KUKA KRL program: rechazoemsinf.src, rechazoemsinf.dat

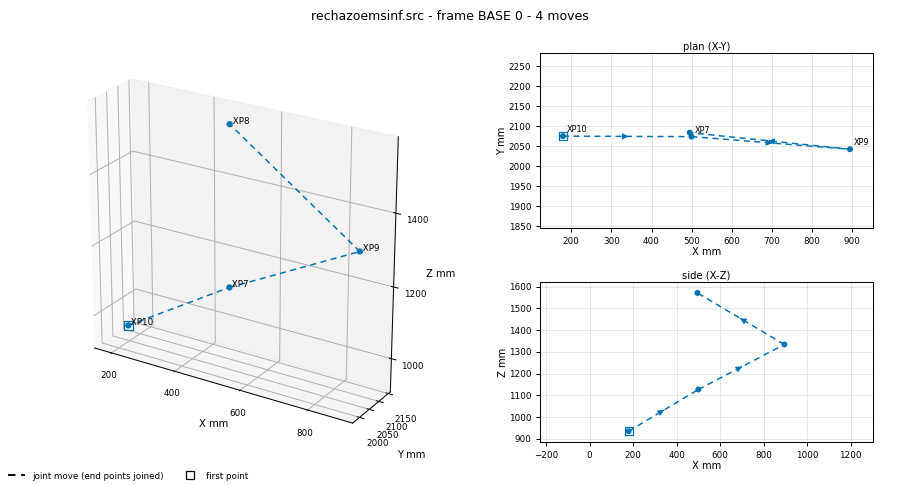
[picture p0: tool path of rechazoemsinf.src in frame BASE 0, 4 of 4 moves have a stored position in this frame; points joined in program order, loops and branches not executed]
--- rechazoemsinf.src ---
&ACCESS RVO1
&REL 33
&COMMENT rechazo ems inferior
&PARAM TEMPLATE = C:\KRC\Roboter\Template\vorgabe
&PARAM EDITMASK = *
DEF RECHAZOEMSINF( )

;================================================
; MODELO   : C-520
; IE GRUPO : 5J
; ESTACION : 85
; ROBOT    : 85r01
; FUNCION  : xxxxxxx
;================================================

;FOLD INI
  ;FOLD BASISTECH INI
    GLOBAL INTERRUPT DECL 3 WHEN $STOPMESS==TRUE DO IR_STOPM ( )
    INTERRUPT ON 3
    BAS (#INITMOV,0 )
  ;ENDFOLD (BASISTECH INI)
;FOLD SPOTTECH INI
;USERSPOT(#INIT)
;ENDFOLD (SPOTTECH INI)
;FOLD GRIPPERTECH INI
USER_GRP(0,DUMMY,DUMMY,GDEFAULT)
INTERRUPT DECL 20 WHEN $FLAG[20]==FALSE DO GRPS(#MON_ERR,20)
;ENDFOLD (GRIPPERTECH INI)
  ;FOLD USER INI
    ;Make your modifications here

  ;ENDFOLD (USER INI)
;ENDFOLD (INI)

I_DATOS_NOK=TRUE

;FOLD PTP P10 CONT Vel=100 % PDAT10 Tool[0] Base[0];%{PE}%R 5.6.13,%MKUKATPBASIS,%CMOVE,%VPTP,%P 1:PTP, 2:P10, 3:C_PTP, 5:100, 7:PDAT10
$BWDSTART=FALSE
PDAT_ACT=PPDAT10
FDAT_ACT=FP10
BAS(#PTP_PARAMS,100)
PTP XP10 C_PTP
;ENDFOLD
;FOLD OUT 18 'LIBERACION AREA 2 ems sup' State=FALSE ;%{PE}%R 5.6.13,%MKUKATPBASIS,%COUT,%VOUTX,%P 2:18, 3:LIBERACION AREA 2 ems sup, 5:FALSE, 6:
$OUT[18]=FALSE
;ENDFOLD
;RECHAZOPOS
;FOLD FORDTECH.Area_Req 4 Safety Position, 0 Return To Home, 0 ;%{PE}%MKUKATPUSER
;Area_Req (4,0,0)

WAIT FOR  ( $IN[20] )
$OUT[20]=FALSE

;ENDFOLD
WAIT SEC 4
;FOLD PTP P7 CONT Vel=30 % PDAT7 Tool[0] Base[0];%{PE}%R 5.6.13,%MKUKATPBASIS,%CMOVE,%VPTP,%P 1:PTP, 2:P7, 3:C_PTP, 5:30, 7:PDAT7
$BWDSTART=FALSE
PDAT_ACT=PPDAT7
FDAT_ACT=FP7
BAS(#PTP_PARAMS,30)
PTP XP7 C_PTP
;ENDFOLD

;FOLD PTP P9 Vel=30 % PDAT9 Tool[0] Base[0];%{PE}%R 5.6.13,%MKUKATPBASIS,%CMOVE,%VPTP,%P 1:PTP, 2:P9, 3:, 5:30, 7:PDAT9
$BWDSTART=FALSE
PDAT_ACT=PPDAT9
FDAT_ACT=FP9
BAS(#PTP_PARAMS,30)
PTP XP9
;ENDFOLD

;FOLD OUT 97 'dedos fuera' State=FALSE ;%{PE}%R 5.6.13,%MKUKATPBASIS,%COUT,%VOUTX,%P 2:97, 3:dedos fuera, 5:FALSE, 6:
$OUT[97]=FALSE
;ENDFOLD
;FOLD OUT 98 'dedos dentro' State=TRUE ;%{PE}%R 5.6.13,%MKUKATPBASIS,%COUT,%VOUTX,%P 2:98, 3:dedos dentro, 5:TRUE, 6:
$OUT[98]=TRUE
;ENDFOLD

;FOLD OUT 89 'pos abrir ip manual' State=TRUE ;%{PE}%R 5.6.13,%MKUKATPBASIS,%COUT,%VOUTX,%P 2:89, 3:pos abrir ip manual, 5:TRUE, 6:
$OUT[89]=TRUE
;ENDFOLD
;FOLD FORDTECH.Tool_Rel 5 ;%{PE}%MKUKATPUSER
TOOL_REL (5)
;ENDFOLD
;FOLD FORDTECH.Tool_Req 5 ;%{PE}%MKUKATPUSER
TOOL_REQ (5)
;ENDFOLD

;FOLD OUT 89 'pos abrir ip manual' State=FALSE ;%{PE}%R 5.6.13,%MKUKATPBASIS,%COUT,%VOUTX,%P 2:89, 3:pos abrir ip manual, 5:FALSE, 6:
$OUT[89]=FALSE
;ENDFOLD
;FOLD OUT 97 'dedos fuera' State=TRUE ;%{PE}%R 5.6.13,%MKUKATPBASIS,%COUT,%VOUTX,%P 2:97, 3:dedos fuera, 5:TRUE, 6:
$OUT[97]=TRUE
;ENDFOLD
;FOLD OUT 98 'dedos dentro' State=FALSE ;%{PE}%R 5.6.13,%MKUKATPBASIS,%COUT,%VOUTX,%P 2:98, 3:dedos dentro, 5:FALSE, 6:
$OUT[98]=FALSE
;ENDFOLD

;FOLD PTP P8 CONT Vel=100 % PDAT8 Tool[0] Base[0];%{PE}%R 5.6.13,%MKUKATPBASIS,%CMOVE,%VPTP,%P 1:PTP, 2:P8, 3:C_PTP, 5:100, 7:PDAT8
$BWDSTART=FALSE
PDAT_ACT=PPDAT8
FDAT_ACT=FP8
BAS(#PTP_PARAMS,100)
PTP XP8 C_PTP
;ENDFOLD
;FOLD FORDTECH.Area_Rel 2 ;%{PE}%MKUKATPUSER
AREA_REL (2)
;ENDFOLD
;FOLD FORDTECH.Area_Rel 3 ;%{PE}%MKUKATPUSER
AREA_REL (3)
;ENDFOLD
;FOLD FORDTECH.Area_Rel 4 ;%{PE}%MKUKATPUSER
AREA_REL (4)
;ENDFOLD
;FOLD FORDTECH.Job_Rdy 4 , 1 ;%{PE}%MKUKATPUSER
JOB_READY (4,1)
;ENDFOLD




END

--- rechazoemsinf.dat ---
&ACCESS RVO1
&REL 33
&COMMENT rechazo ems inferior
&PARAM TEMPLATE = C:\KRC\Roboter\Template\vorgabe
&PARAM EDITMASK = *
DEFDAT  RECHAZOEMSINF
;FOLD EXTERNAL DECLARATIONS;%{PE}%MKUKATPBASIS,%CEXT,%VCOMMON,%P
;FOLD GRIPPERTECH EXT
EXT  H50 (INT  :IN,INT  :IN,INT  :IN,GRP_TYP  :IN )
;ENDFOLD (GRIPPERTECH EXT)
;FOLD SPOTTECH EXT
EXT  USERSPOT (S_COMMAND  :IN,SPOT_TYPE  :IN )
;ENDFOLD (SPOTTECH EXT)
;FOLD BASISTECH EXT;%{PE}%MKUKATPBASIS,%CEXT,%VEXT,%P
EXT  BAS (BAS_COMMAND  :IN,REAL  :IN )
DECL INT SUCCESS
;ENDFOLD (BASISTECH EXT)
;FOLD USER EXT;%{E}%MKUKATPUSER,%CEXT,%VEXT,%P
;Make here your modifications

;ENDFOLD (USER EXT)
;ENDFOLD (EXTERNAL DECLARATIONS)
DECL BASIS_SUGG_T LAST_BASIS={POINT1[] "P10                     ",POINT2[] "P10                     ",CP_PARAMS[] "CPDAT0                  ",PTP_PARAMS[] "PDAT10                  ",CONT[] "C_PTP                   ",CP_VEL[] "2.0                     ",PTP_VEL[] "100                     ",SYNC_PARAMS[] "SYNCDAT                 ",SPL_NAME[] "S0                      "}
DECL PDAT PPDAT0={VEL 100.0,ACC 100.0,APO_DIST 100.0}
DECL E6POS XP0={X 1811.52502,Y -400.592712,Z 796.957886,A -63.3204193,B 28.7300301,C -159.576996,S 2,T 10,E1 0.0,E2 0.0,E3 0.0,E4 0.0,E5 0.0,E6 0.0}
DECL FDAT FP0={TOOL_NO 1,BASE_NO 0,IPO_FRAME #BASE,POINT2[] " ",TQ_STATE FALSE}
DECL PDAT PPDAT1={VEL 100.0,ACC 100.0,APO_DIST 100.0,APO_MODE #CPTP}
DECL E6POS XP1={X 141.040298,Y -131.536896,Z -626.476685,A -0.01522478,B 7.10692596,C 0.110732399,S 2,T 3,E1 0.0,E2 0.0,E3 0.0,E4 0.0,E5 0.0,E6 0.0}
DECL FDAT FP1={TOOL_NO 3,BASE_NO 8,IPO_FRAME #BASE,POINT2[] " ",TQ_STATE FALSE}
DECL PDAT PPDAT2={VEL 100.0,ACC 100.0,APO_DIST 100.0,APO_MODE #CPTP}
DECL E6POS XP2={X 1145.12195,Y 865.575378,Z 1562.22705,A -24.1379299,B -0.725280404,C -90.2146072,S 2,T 2,E1 0.0,E2 0.0,E3 0.0,E4 0.0,E5 0.0,E6 0.0}
DECL FDAT FP2={TOOL_NO 3,BASE_NO 0,IPO_FRAME #BASE,POINT2[] " ",TQ_STATE FALSE}
DECL PDAT PPDAT3={VEL 100.0,ACC 100.0,APO_DIST 100.0,APO_MODE #CPTP}
DECL E6POS XP3={X 1888.578,Y 938.442871,Z 1603.72998,A -59.9518318,B -1.77833796,C -87.043541,S 2,T 2,E1 0.0,E2 0.0,E3 0.0,E4 0.0,E5 0.0,E6 0.0}
DECL FDAT FP3={TOOL_NO 3,BASE_NO 0,IPO_FRAME #BASE,POINT2[] " ",TQ_STATE FALSE}
DECL PDAT PPDAT4={VEL 100.0,ACC 100.0,APO_DIST 100.0,APO_MODE #CPTP}
DECL E6POS XP4={X 2768.47705,Y 6.94654799,Z 2006.30298,A -150.0289,B 15.6658697,C -84.9255676,S 2,T 43,E1 0.0,E2 0.0,E3 0.0,E4 0.0,E5 0.0,E6 0.0}
DECL FDAT FP4={TOOL_NO 3,BASE_NO 0,IPO_FRAME #BASE,POINT2[] " ",TQ_STATE FALSE}
DECL E6POS XP5={X 690.610596,Y 1039.49902,Z 547.695374,A 1.02792203,B -0.0946048573,C -89.774292,S 2,T 11,E1 0.0,E2 0.0,E3 0.0,E4 0.0,E5 0.0,E6 0.0}
DECL FDAT FP5={TOOL_NO 3,BASE_NO 0,IPO_FRAME #BASE,POINT2[] " ",TQ_STATE FALSE}
DECL PDAT PPDAT5={VEL 100.0,ACC 100.0,APO_DIST 100.0,APO_MODE #CPTP}
DECL E6POS XP6={X 1195.56702,Y 865.034424,Z 1032.25696,A -14.0337496,B 8.53373337,C -49.2474098,S 2,T 10,E1 0.0,E2 0.0,E3 0.0,E4 0.0,E5 0.0,E6 0.0}
DECL FDAT FP6={TOOL_NO 3,BASE_NO 0,IPO_FRAME #BASE,POINT2[] " ",TQ_STATE FALSE}
DECL PDAT PPDAT6={VEL 100.0,ACC 100.0,APO_DIST 100.0,APO_MODE #CPTP}
DECL E6POS XP7={X 499.745209,Y 2073.84009,Z 1127.026,A -0.35774979,B 45.6510086,C 179.642807,S 2,T 11,E1 0.0,E2 0.0,E3 0.0,E4 0.0,E5 0.0,E6 0.0}
DECL FDAT FP7={TOOL_NO 0,BASE_NO 0,IPO_FRAME #BASE,POINT2[] " ",TQ_STATE FALSE}
DECL PDAT PPDAT7={VEL 100.0,ACC 100.0,APO_DIST 100.0,APO_MODE #CPTP}
DECL E6POS XP8={X 495.390503,Y 2083.77197,Z 1570.86499,A 13.1525097,B 38.8060799,C -160.305206,S 2,T 11,E1 0.0,E2 0.0,E3 0.0,E4 0.0,E5 0.0,E6 0.0}
DECL FDAT FP8={TOOL_NO 0,BASE_NO 0,IPO_FRAME #BASE,POINT2[] " ",TQ_STATE FALSE}
DECL PDAT PPDAT8={VEL 100.0,ACC 100.0,APO_DIST 100.0,APO_MODE #CPTP}
DECL PDAT PPDAT9={VEL 100.0,ACC 100.0,APO_DIST 100.0}
DECL E6POS XP9={X 895.210388,Y 2042.41199,Z 1333.90002,A 3.05633497,B 48.7101097,C -175.618301,S 2,T 11,E1 0.0,E2 0.0,E3 0.0,E4 0.0,E5 0.0,E6 0.0}
DECL FDAT FP9={TOOL_NO 0,BASE_NO 0,IPO_FRAME #BASE,POINT2[] " ",TQ_STATE FALSE}
DECL E6POS XP10={X 179.160904,Y 2075.0249,Z 935.252686,A -0.490047991,B 45.5180817,C 179.520294,S 2,T 11,E1 0.0,E2 0.0,E3 0.0,E4 0.0,E5 0.0,E6 0.0}
DECL FDAT FP10={TOOL_NO 0,BASE_NO 0,IPO_FRAME #BASE,POINT2[] " ",TQ_STATE FALSE}
DECL PDAT PPDAT10={VEL 100.0,ACC 100.0,APO_DIST 100.0,APO_MODE #CPTP}
ENDDAT
